FUNCTION_BLOCK Lincon
VAR_INPUT
	Enable:BOOL; (**)
	Input:REAL; (**)
	Multiplier:REAL; (**)
	Divisor:REAL; (**)
	Offset:REAL; (**)
END_VAR
VAR_OUTPUT
	Out:REAL; (**)
END_VAR
VAR
END_VAR
VAR
	Mul_r:REAL;
	Div_r:REAL;
	In_r:REAL;
	Out_r:REAL;
	Err_b:BOOL;
	tempMemAddr:REAL;
END_VAR

{warning 'TODO: Two places need the equivalent of %S18 placed here. Be sure to delete the tempMemAddr var when you are done.'}
VAR // added by the converter: edge detectors and wires of the graphical bodies
    _w1, _w2, _w9, _w11, _w12, _w13, _w15 : BOOL;
    _w3, _w4, _w5, _w6, _w7, _w8, _w14 : REAL;
    _w10, _w16 : ANY;
END_VAR

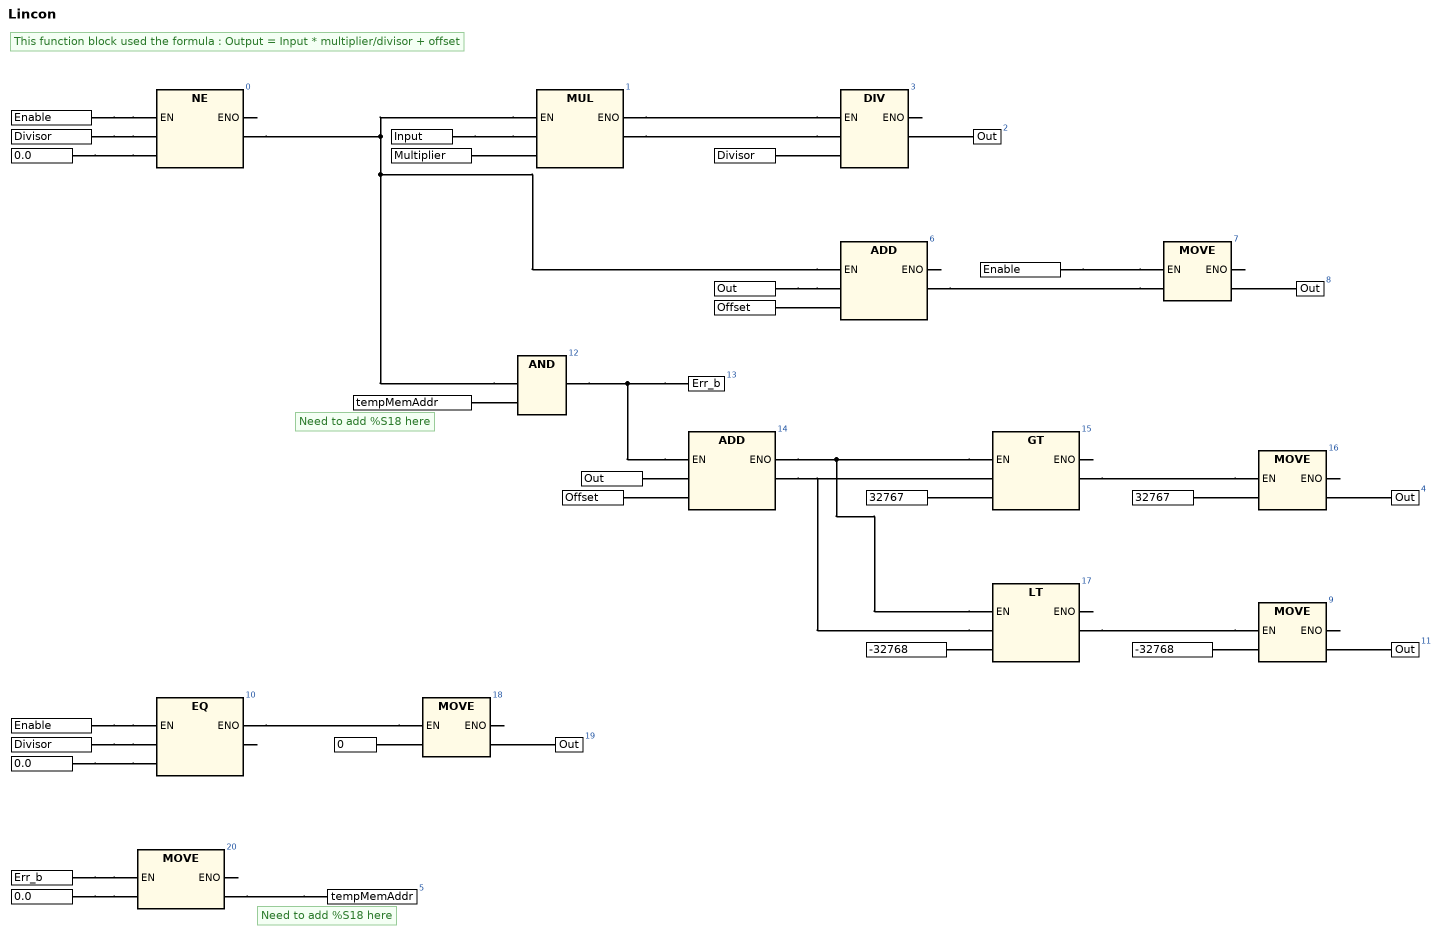
// This function block used the formula : Output = Input * multiplier/divisor + offset
IF Enable THEN _w1 := Divisor <> 0.0; END_IF
_w2 := _w1;
IF _w2 THEN _w3 := Input * Multiplier; END_IF
Out := _w4;
IF _w2 THEN _w4 := _w3 / Divisor; END_IF
Out := _w5;
// Need to add %S18 here
tempMemAddr := _w6;
IF _w1 THEN _w7 := Out + Offset; END_IF
IF Enable THEN _w8 := _w7; END_IF
Out := _w8;
IF _w9 THEN _w10 := -32768; END_IF
_w11 := Enable;
IF _w11 THEN (* Divisor = 0.0; result not used *) END_IF
Out := _w10;
_w12 := _w1 AND tempMemAddr;
Err_b := _w12;
// Need to add %S18 here
_w13 := _w12;
IF _w13 THEN _w14 := Out + Offset; END_IF
IF _w13 THEN _w15 := _w14 > 32767; END_IF
IF _w15 THEN _w5 := 32767; END_IF
IF _w13 THEN _w9 := _w14 < -32768; END_IF
IF _w11 THEN _w16 := 0; END_IF
Out := _w16;
IF Err_b THEN _w6 := 0.0; END_IF

END_FUNCTION_BLOCK

(* stored: Version 1.1.0.1, ProductVersion 3.1.4024.0
   POU Lincon: Id {5dfe4370-8e73-4ee7-bda7-e92777189b08}, SpecialFunc None *)
